PROGRAM Main
VAR
END_VAR

END_PROGRAM

(* stored: Version 1.1.0.1, ProductVersion 3.1.4024.0
   POU Main: Id {70235fb6-3685-4fb1-a11c-2aa1f01d1de9}, SpecialFunc None *)
